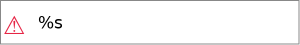
VISUALIZATION Uc_Component  // 300x45
    Rectangle (35,0 265x45), "%s", text variable: stVisu.sName
        p55702900: sel(stvisu.bEnable,colBlack50, colBlack)
    Rectangle (0,5 35x40), "⚠", text variable: stVisu.sName, invisible if: NOT stVisu.bError
        OnMouseClick: execute { stvisu.bReset := TRUE; }
END_VISUALIZATION

(* stored: Version 1.1.0.1
   Visu Uc_Component: Id {3a5154ad-bc39-42c5-ba13-867188883eff} *)
